Universal Robots URScript: util_script.script

# General UR Utilities
# File: util_script.script
# Version 1.0
# Programmer: Ned Lecky

# Send CRLF out the socket
def socket_send_crlf():
  socket_send_byte(13)
  socket_send_byte(10)
end

# Send LF out the socket
def socket_send_lf():
  socket_send_byte(10)
end

# Conversion (RPY(deg) to AxisAngle)
def RPY_to_AxisAngle(R):
  Rx = d2r(R[3]) / 2.0
  Ry = d2r(R[4]) / 2.0
  Rz = d2r(R[5]) / 2.0

  Cx = cos(Rx)
  Sx = sin(Rx)
  Cy = cos(Ry)
  Sy = sin(Ry)
  Cz = cos(Rz)
  Sz = sin(Rz)

  Angle = 2.0 * acos(Cx * Cy * Cz + Sx * Sy * Sz)
  x = Sx * Cy * Cz - Cx * Sy * Sz
  y = Cx * Sy * Cz + Sx * Cy * Sz
  z = -Sx * Sy * Cz + Cx * Cy * Sz
  Norm = sqrt(x * x + y * y + z * z)
  if norm(Norm) < 1e-4:
    Ax = 0
    Ay = 0
    Az = 0
  else:
    Ratio = Angle / Norm
    Ax = x * Ratio
    Ay = y * Ratio
    Az = z * Ratio
  end
  Ans = p[R[0], R[1], R[2], Ax, Ay, Az]

  return Ans
end

# Conversion (AxisAngle to RPY)
def AxisAngle_to_RPY(R):
  Rx = R[3]
  Ry = R[4]
  Rz = R[5]

  Angle = sqrt(Rx * Rx + Ry * Ry + Rz * Rz)
  if Angle < 1e-4:
    x = 0
    y = 0
    z = 1
  else:
    x = Rx / Angle
    y = Ry / Angle
    z = Rz / Angle
  end
  S = sin(Angle)
  C = cos(Angle)
  T = 1 - C

  r11 = T * x * x + C
  r12 = T * x * y - S * z
  r13 = T * x * z + S * y
  r21 = T * x * y + S * z
  r22 = T * y * y + C
  r23 = T * y * z - S * x
  r31 = T * x * z - S * y
  r32 = T * y * z + S * x
  r33 = T * z * z + C

  if r31 > 1:
    r31 = 1
  elif r31 < -1:
    r31 = -1
  end

  Ay = asin(-r31)
  if Ay > d2r(89.9):
    sinAxMinusAz = (r12 - r23) / (1 - r31)
    cosAxMinusAz = (r13 + r22) / (1 - r31)
    Ax = atan2(sinAxMinusAz, cosAxMinusAz)
    Az = 0
  elif Ay < d2r(-89.9):
    sinAxPlusAz = (-r12 - r23) / (1 + r31)
    cosAxPlusAz = (-r13 + r22) / (1 + r31)
    Ax = atan2(sinAxPlusAz, cosAxPlusAz)
    Az = 0
  else:
    Ax = atan2(r32, r33)
    Az = atan2(r21, r11)
  end

  Ans = p[R[0], R[1], R[2], r2d(Ax), r2d(Ay), r2d(Az)]

  return Ans
end

# Get position in RPY coordinate
def get_actual_tcp_pose_RPY():
  p = get_actual_tcp_pose()
  p2 = AxisAngle_to_RPY(p)
  return p2
end

# movel in RPY coordinates
def movel_RPY(p, accel, speed):
  p1 = RPY_to_AxisAngle(p)
  movel(p1, accel, speed)
end

# movej in RPY coordinates
def movej_RPY(p, accel, speed):
  p1 = RPY_to_AxisAngle(p)
  movej(p1, accel, speed)
end

# Add position
def pose_add_RPY(V1, V2):
  A0 = V1[0] + V2[0]
  A1 = V1[1] + V2[1]
  A2 = V1[2] + V2[2]
  A3 = V1[3] + V2[3]
  A4 = V1[4] + V2[4]
  A5 = V1[5] + V2[5]
  A = p[A0, A1, A2, A3, A4, A5]

  return A
end

# Send 6-vectors back to socket as [n,n,n,n,n,n]
def return_vector(p):
  socket_send_string("[")
  i = 0
  while i < 6:
    if i > 0:
      socket_send_string(",")
    end
    socket_send_string(p[i])
    i = i + 1
  end
  socket_send_string("]")
end

# Send 6-element position back to socket as:
#   (isPose=False) name=[n,n,n,n,n,n]
#   (isPose=True)name=p[n,n,n,n,n,n]
def return_position(name, isPose, p):
  socket_send_string(name)
  socket_send_string("=")
  if isPose == True:
    socket_send_string("p")
  end
  return_vector(p)
  socket_send_lf()
end

# Return a 6-element vector as a pose name=p[.....]
def return_pose(name, p):
  return_position(name, True, p)
end

# Return a 6-element vector as joint angles name=[.....]
def return_joints(name, p):
  return_position(name, False, p)
end
